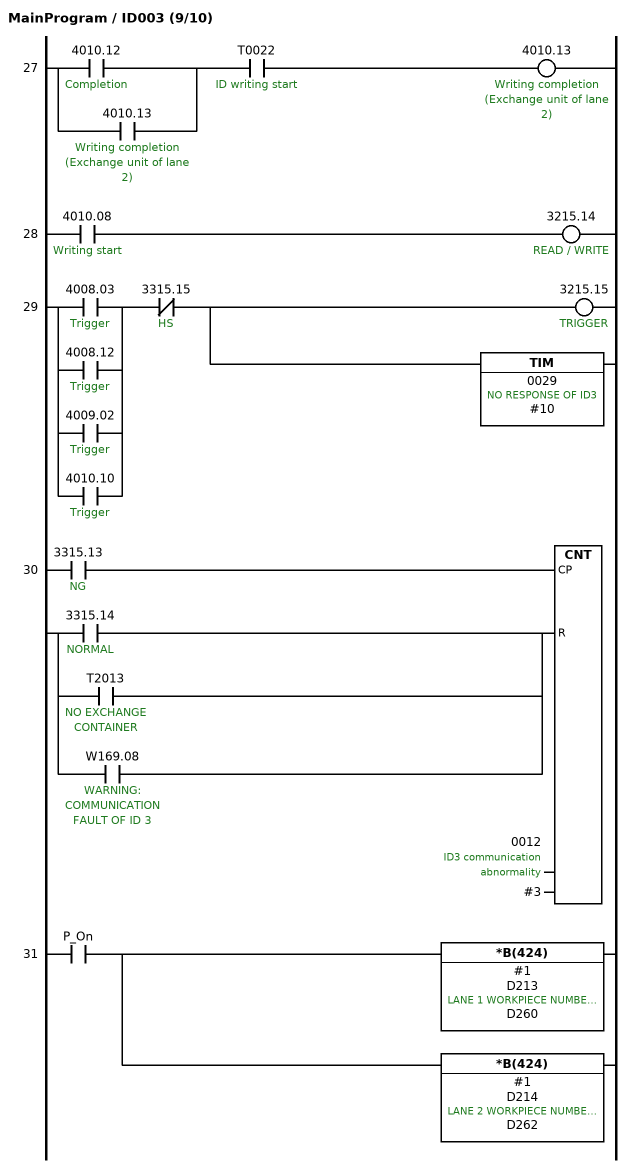
; [picture p48: MainProgram / ID003, rungs 27-31]
; rung 27
LD 4010.12  ; Completion
OR 4010.13  ; Writing completion (Exchange unit of lane 2)
AND T0022  ; ID writing start
OUT 4010.13  ; Writing completion (Exchange unit of lane 2)
; rung 28
LD 4010.08  ; Writing start
OUT 3215.14  ; READ / WRITE
; rung 29
LD 4008.03  ; Trigger
OR 4008.12  ; Trigger
OR 4009.02  ; Trigger
OR 4010.10  ; Trigger
ANDNOT 3315.15  ; HS
OUT 3215.15  ; TRIGGER
TIM 0029 #10  ; NO RESPONSE OF ID3
; rung 30
LD 3315.13  ; NG
LD 3315.14  ; NORMAL
OR T2013  ; NO EXCHANGE CONTAINER
OR W169.08  ; WARNING:COMMUNICATION FAULT OF ID 3
CNT 0012 #3  ; ID3 communication abnormality
; rung 31
LD P_On
*B(424) #1 D213 D260  ; LANE 1 WORKPIECE NUMBER DISPLAY
*B(424) #1 D214 D262  ; LANE 2 WORKPIECE NUMBER DISPLAY

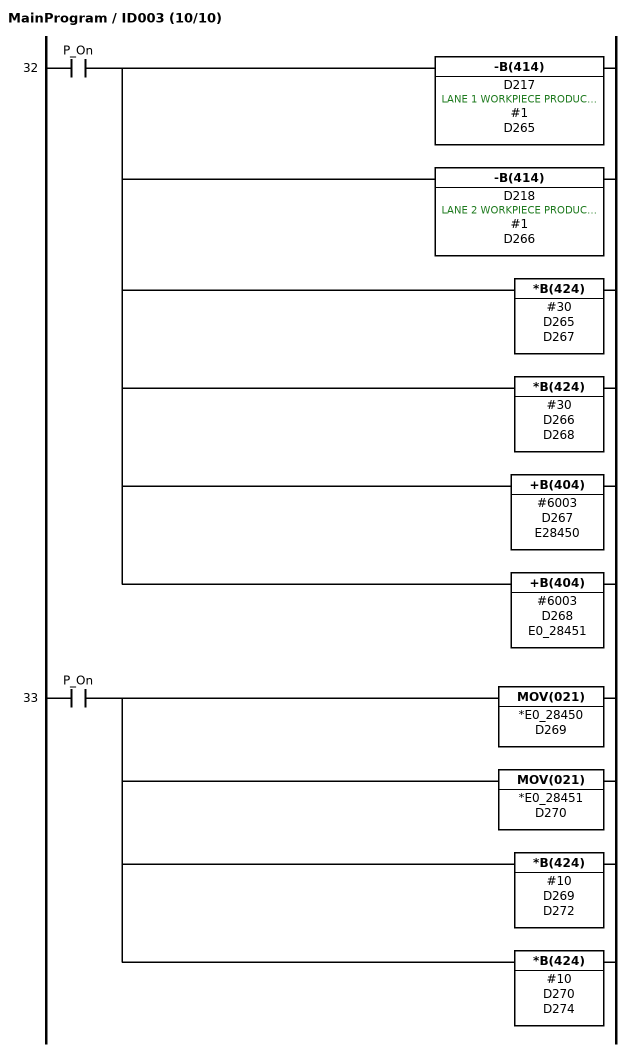
; rung 32
LD P_On
-B(414) D217 #1 D265  ; LANE 1 WORKPIECE PRODUCT NUMBER
-B(414) D218 #1 D266  ; LANE 2 WORKPIECE PRODUCT NUMBER
*B(424) #30 D265 D267
*B(424) #30 D266 D268
+B(404) #6003 D267 E28450
+B(404) #6003 D268 E0_28451
; rung 33
LD P_On
MOV(021) *E0_28450 D269
MOV(021) *E0_28451 D270
*B(424) #10 D269 D272
*B(424) #10 D270 D274

### Section ID004

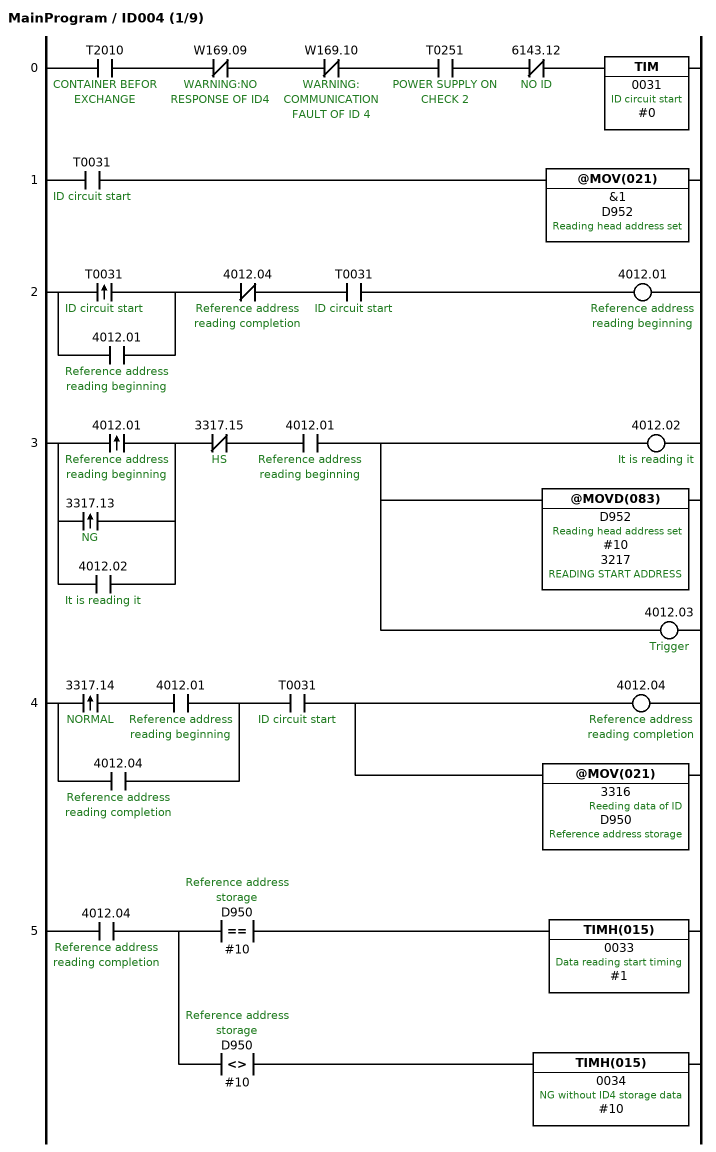
; rung 0
LD T2010  ; CONTAINER BEFOR EXCHANGE
ANDNOT W169.09  ; WARNING:NO RESPONSE OF ID4
ANDNOT W169.10  ; WARNING:COMMUNICATION FAULT OF ID 4
AND T0251  ; POWER SUPPLY ON CHECK 2
ANDNOT 6143.12  ; NO ID
TIM 0031 #0  ; ID circuit start
; rung 1
LD T0031  ; ID circuit start
@MOV(021) &1 D952  ; Reading head address set
; rung 2
@LD T0031  ; ID circuit start
OR 4012.01  ; Reference address reading beginning
ANDNOT 4012.04  ; Reference address reading completion
AND T0031  ; ID circuit start
OUT 4012.01  ; Reference address reading beginning
; rung 3
@LD 4012.01  ; Reference address reading beginning
@OR 3317.13  ; NG
OR 4012.02  ; It is reading it
ANDNOT 3317.15  ; HS
AND 4012.01  ; Reference address reading beginning
OUT 4012.02  ; It is reading it
@MOVD(083) D952 #10 3217  ; Reading head address set, READING START ADDRESS
OUT 4012.03  ; Trigger
; rung 4
@LD 3317.14  ; NORMAL
AND 4012.01  ; Reference address reading beginning
OR 4012.04  ; Reference address reading completion
AND T0031  ; ID circuit start
OUT 4012.04  ; Reference address reading completion
@MOV(021) 3316 D950  ; Reeding data of ID, Reference address storage
; rung 5
LD 4012.04  ; Reference address reading completion
OUT TR0
AND=(300) D950 #10  ; Reference address storage
TIMH(015) 0033 #1  ; Data reading start timing
LD TR0
AND<>(305) D950 #10  ; Reference address storage
TIMH(015) 0034 #10  ; NG without ID4 storage data

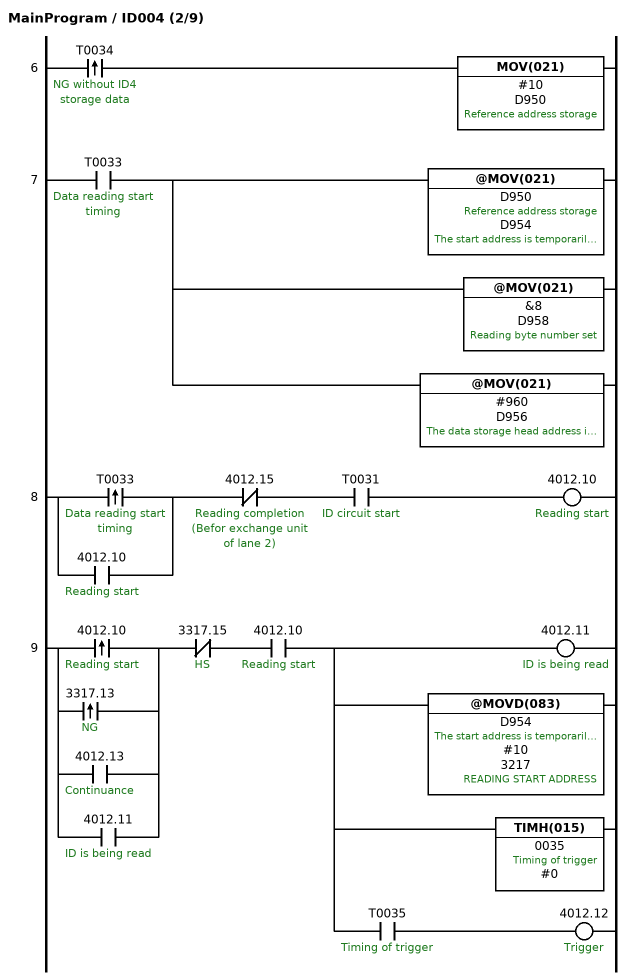
; rung 6
@LD T0034  ; NG without ID4 storage data
MOV(021) #10 D950  ; Reference address storage
; rung 7
LD T0033  ; Data reading start timing
@MOV(021) D950 D954  ; Reference address storage, The start address is temporarily memorized
@MOV(021) &8 D958  ; Reading byte number set
@MOV(021) #960 D956  ; The data storage head address is memorized
; rung 8
@LD T0033  ; Data reading start timing
OR 4012.10  ; Reading start
ANDNOT 4012.15  ; Reading completion (Befor exchange unit of lane 2)
AND T0031  ; ID circuit start
OUT 4012.10  ; Reading start
; rung 9
@LD 4012.10  ; Reading start
@OR 3317.13  ; NG
OR 4012.13  ; Continuance
OR 4012.11  ; ID is being read
ANDNOT 3317.15  ; HS
AND 4012.10  ; Reading start
OUT 4012.11  ; ID is being read
@MOVD(083) D954 #10 3217  ; The start address is temporarily memorized, READING START ADDRESS
TIMH(015) 0035 #0  ; Timing of trigger
AND T0035  ; Timing of trigger
OUT 4012.12  ; Trigger

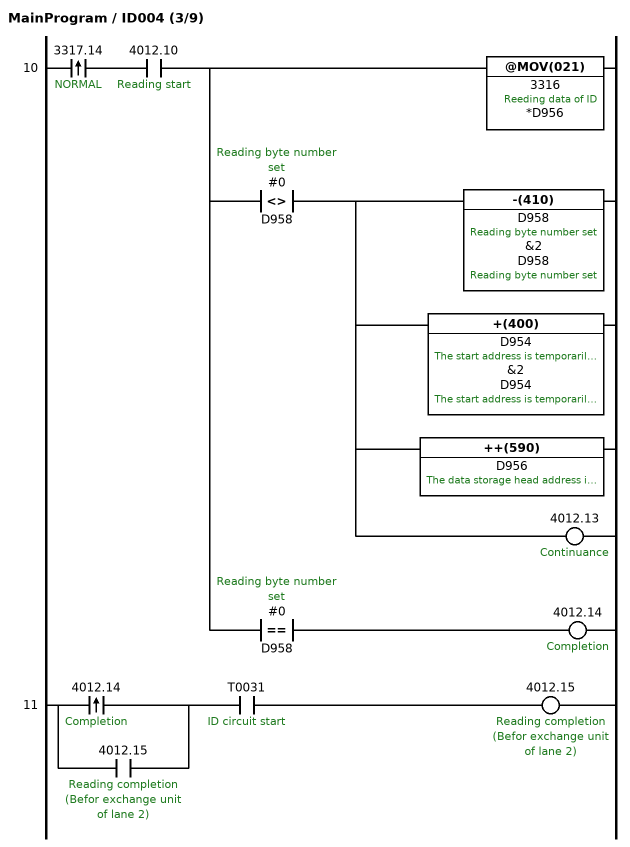
; rung 10
@LD 3317.14  ; NORMAL
AND 4012.10  ; Reading start
OUT TR0
@MOV(021) 3316 *D956  ; Reeding data of ID
AND<>(305) #0 D958  ; Reading byte number set
-(410) D958 &2 D958  ; Reading byte number set
+(400) D954 &2 D954  ; The start address is temporarily memorized
++(590) D956  ; The data storage head address is memorized
OUT 4012.13  ; Continuance
LD TR0
AND=(300) #0 D958  ; Reading byte number set
OUT 4012.14  ; Completion
; rung 11
@LD 4012.14  ; Completion
OR 4012.15  ; Reading completion (Befor exchange unit of lane 2)
AND T0031  ; ID circuit start
OUT 4012.15  ; Reading completion (Befor exchange unit of lane 2)

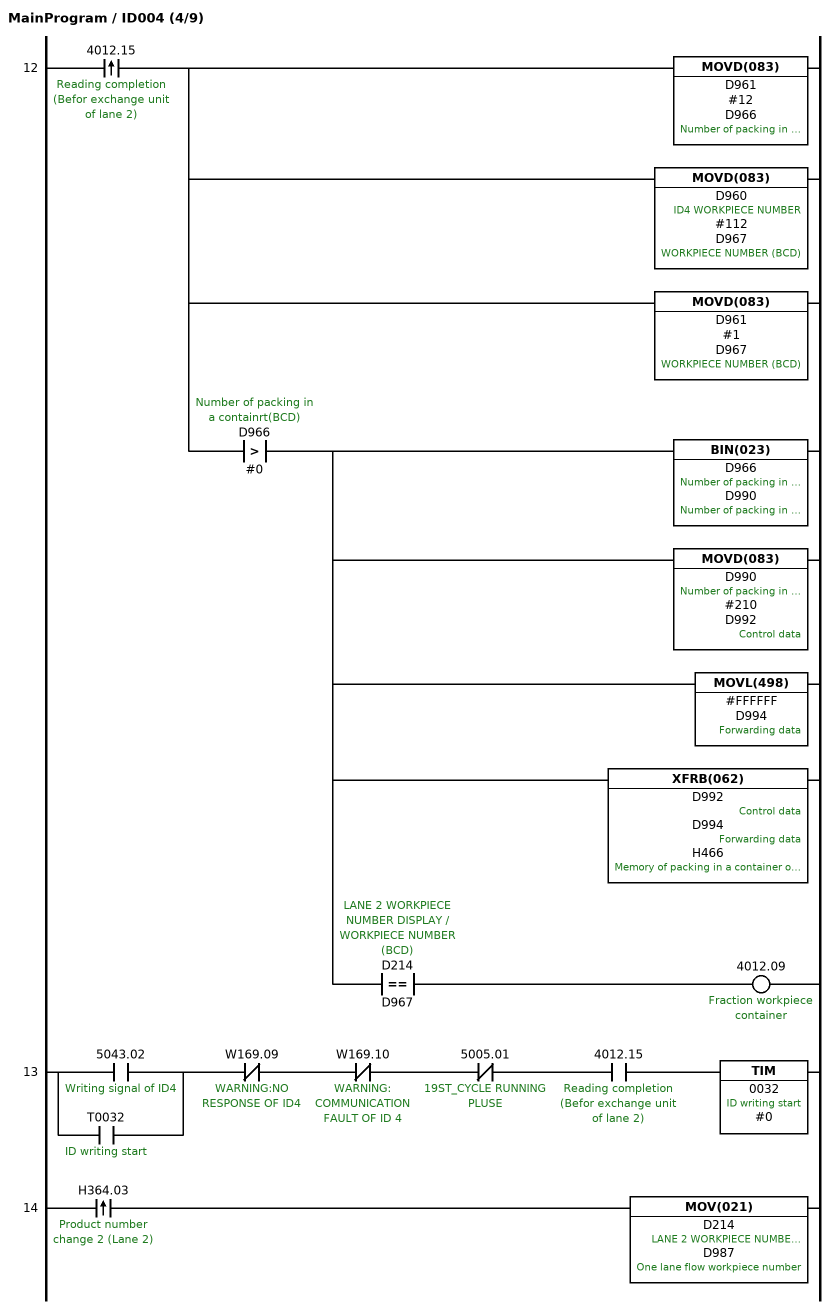
; rung 12
@LD 4012.15  ; Reading completion (Befor exchange unit of lane 2)
MOVD(083) D961 #12 D966  ; Number of packing in a containrt(BCD)
MOVD(083) D960 #112 D967  ; ID4 WORKPIECE NUMBER, WORKPIECE NUMBER (BCD)
MOVD(083) D961 #1 D967  ; WORKPIECE NUMBER (BCD)
AND>(320) D966 #0  ; Number of packing in a containrt(BCD)
BIN(023) D966 D990  ; Number of packing in a containrt(BCD), Number of packing in a containrt(BIN)
MOVD(083) D990 #210 D992  ; Number of packing in a containrt(BIN), Control data
MOVL(498) #FFFFFF D994  ; Forwarding data
XFRB(062) D992 D994 H466  ; Control data, Forwarding data, Memory of packing in a container of lane 2 (container befor exchange)
AND=(300) D214 D967  ; LANE 2 WORKPIECE NUMBER DISPLAY, WORKPIECE NUMBER (BCD)
OUT 4012.09  ; Fraction workpiece container
; rung 13
LD 5043.02  ; Writing signal of ID4
OR T0032  ; ID writing start
ANDNOT W169.09  ; WARNING:NO RESPONSE OF ID4
ANDNOT W169.10  ; WARNING:COMMUNICATION FAULT OF ID 4
ANDNOT 5005.01  ; 19ST_CYCLE RUNNING PLUSE
AND 4012.15  ; Reading completion (Befor exchange unit of lane 2)
TIM 0032 #0  ; ID writing start
; rung 14
@LD H364.03  ; Product number change 2 (Lane 2)
MOV(021) D214 D987  ; LANE 2 WORKPIECE NUMBER DISPLAY, One lane flow workpiece number

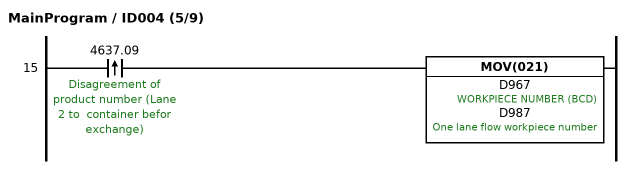
; rung 15
@LD 4637.09  ; Disagreement of product number (Lane 2 to  container befor exchange)
MOV(021) D967 D987  ; WORKPIECE NUMBER (BCD), One lane flow workpiece number

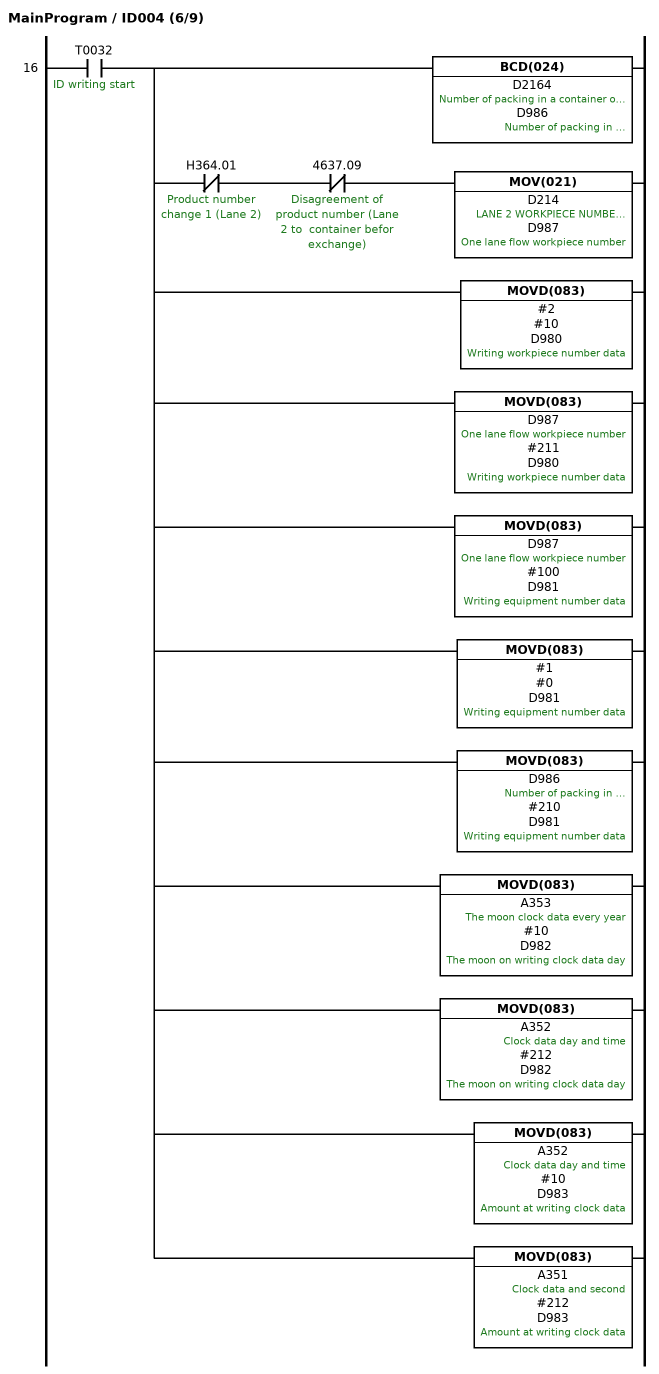
; rung 16
LD T0032  ; ID writing start
OUT TR0
BCD(024) D2164 D986  ; Number of packing in a container of lane 2 (container before exchange)(BIN), Number of packing in a containrt(BCD)
ANDNOT H364.01  ; Product number change 1 (Lane 2)
ANDNOT 4637.09  ; Disagreement of product number (Lane 2 to  container befor exchange)
MOV(021) D214 D987  ; LANE 2 WORKPIECE NUMBER DISPLAY, One lane flow workpiece number
LD TR0
MOVD(083) #2 #10 D980  ; Writing workpiece number data
MOVD(083) D987 #211 D980  ; One lane flow workpiece number, Writing workpiece number data
MOVD(083) D987 #100 D981  ; One lane flow workpiece number, Writing equipment number data
MOVD(083) #1 #0 D981  ; Writing equipment number data
MOVD(083) D986 #210 D981  ; Number of packing in a containrt(BCD), Writing equipment number data
MOVD(083) A353 #10 D982  ; The moon clock data every year, The moon on writing clock data day
MOVD(083) A352 #212 D982  ; Clock data day and time, The moon on writing clock data day
MOVD(083) A352 #10 D983  ; Clock data day and time, Amount at writing clock data
MOVD(083) A351 #212 D983  ; Clock data and second, Amount at writing clock data

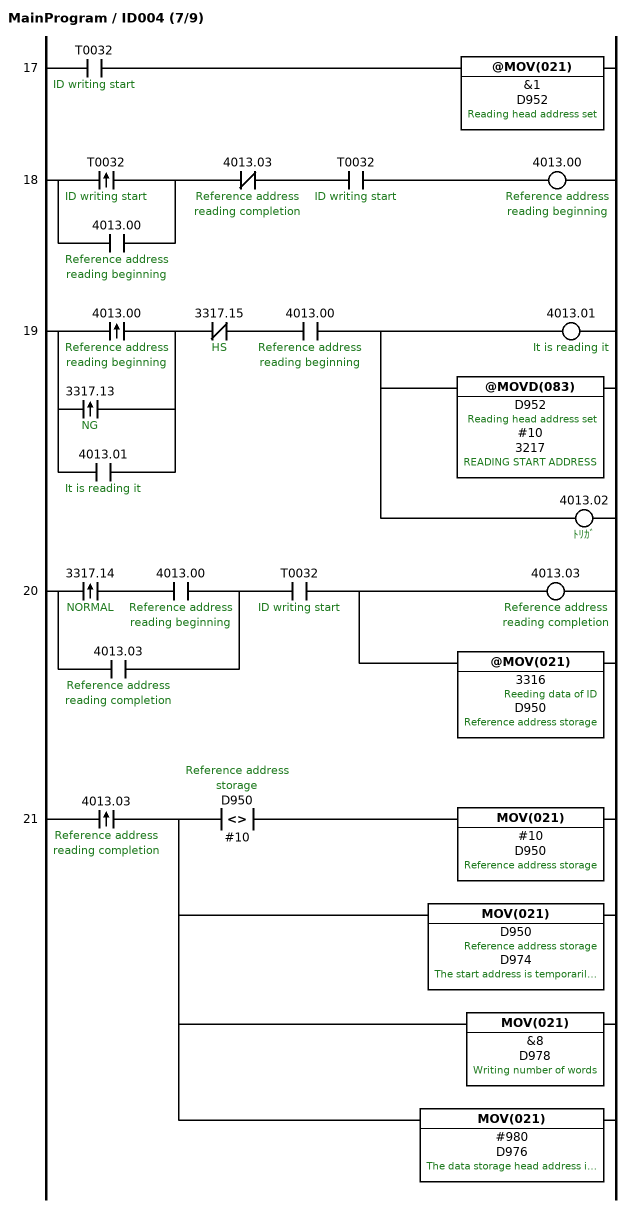
; rung 17
LD T0032  ; ID writing start
@MOV(021) &1 D952  ; Reading head address set
; rung 18
@LD T0032  ; ID writing start
OR 4013.00  ; Reference address reading beginning
ANDNOT 4013.03  ; Reference address reading completion
AND T0032  ; ID writing start
OUT 4013.00  ; Reference address reading beginning
; rung 19
@LD 4013.00  ; Reference address reading beginning
@OR 3317.13  ; NG
OR 4013.01  ; It is reading it
ANDNOT 3317.15  ; HS
AND 4013.00  ; Reference address reading beginning
OUT 4013.01  ; It is reading it
@MOVD(083) D952 #10 3217  ; Reading head address set, READING START ADDRESS
OUT 4013.02  ; ﾄﾘｶﾞ
; rung 20
@LD 3317.14  ; NORMAL
AND 4013.00  ; Reference address reading beginning
OR 4013.03  ; Reference address reading completion
AND T0032  ; ID writing start
OUT 4013.03  ; Reference address reading completion
@MOV(021) 3316 D950  ; Reeding data of ID, Reference address storage
; rung 21
@LD 4013.03  ; Reference address reading completion
OUT TR0
AND<>(305) D950 #10  ; Reference address storage
MOV(021) #10 D950  ; Reference address storage
LD TR0
MOV(021) D950 D974  ; Reference address storage, The start address is temporarily memorized
MOV(021) &8 D978  ; Writing number of words
MOV(021) #980 D976  ; The data storage head address is memorized

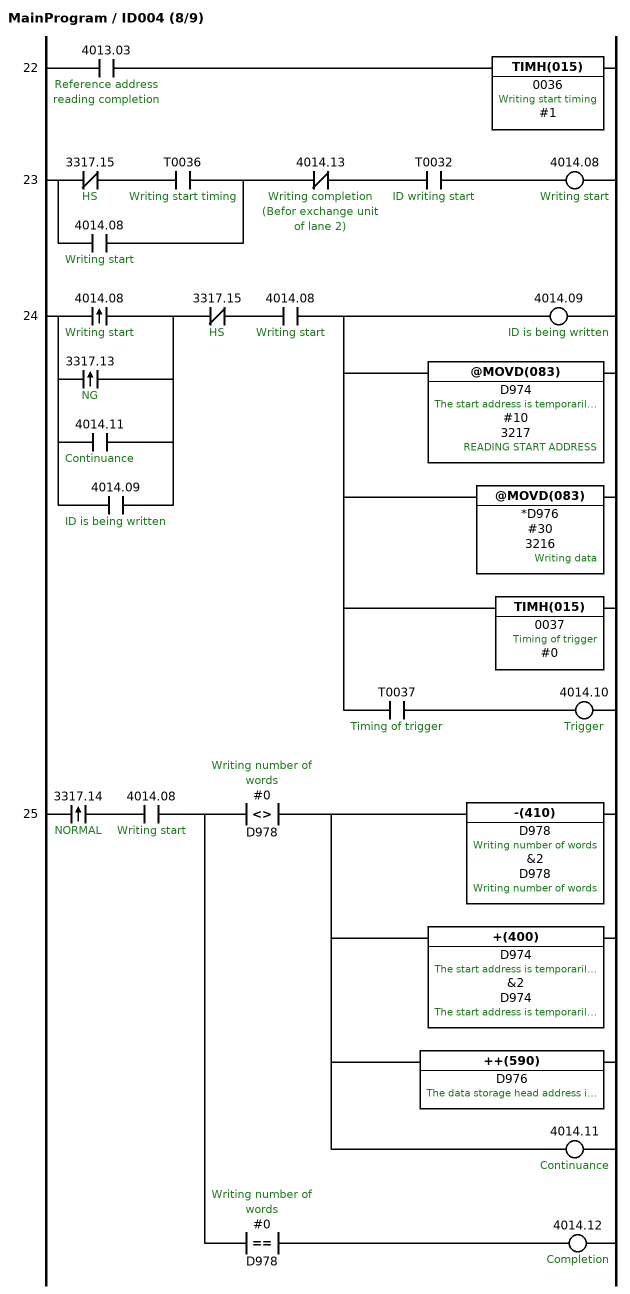
; rung 22
LD 4013.03  ; Reference address reading completion
TIMH(015) 0036 #1  ; Writing start timing
; rung 23
LDNOT 3317.15  ; HS
AND T0036  ; Writing start timing
OR 4014.08  ; Writing start
ANDNOT 4014.13  ; Writing completion (Befor exchange unit of lane 2)
AND T0032  ; ID writing start
OUT 4014.08  ; Writing start
; rung 24
@LD 4014.08  ; Writing start
@OR 3317.13  ; NG
OR 4014.11  ; Continuance
OR 4014.09  ; ID is being written
ANDNOT 3317.15  ; HS
AND 4014.08  ; Writing start
OUT 4014.09  ; ID is being written
@MOVD(083) D974 #10 3217  ; The start address is temporarily memorized, READING START ADDRESS
@MOVD(083) *D976 #30 3216  ; Writing data
TIMH(015) 0037 #0  ; Timing of trigger
AND T0037  ; Timing of trigger
OUT 4014.10  ; Trigger
; rung 25
@LD 3317.14  ; NORMAL
AND 4014.08  ; Writing start
OUT TR0
AND<>(305) #0 D978  ; Writing number of words
-(410) D978 &2 D978  ; Writing number of words
+(400) D974 &2 D974  ; The start address is temporarily memorized
++(590) D976  ; The data storage head address is memorized
OUT 4014.11  ; Continuance
LD TR0
AND=(300) #0 D978  ; Writing number of words
OUT 4014.12  ; Completion

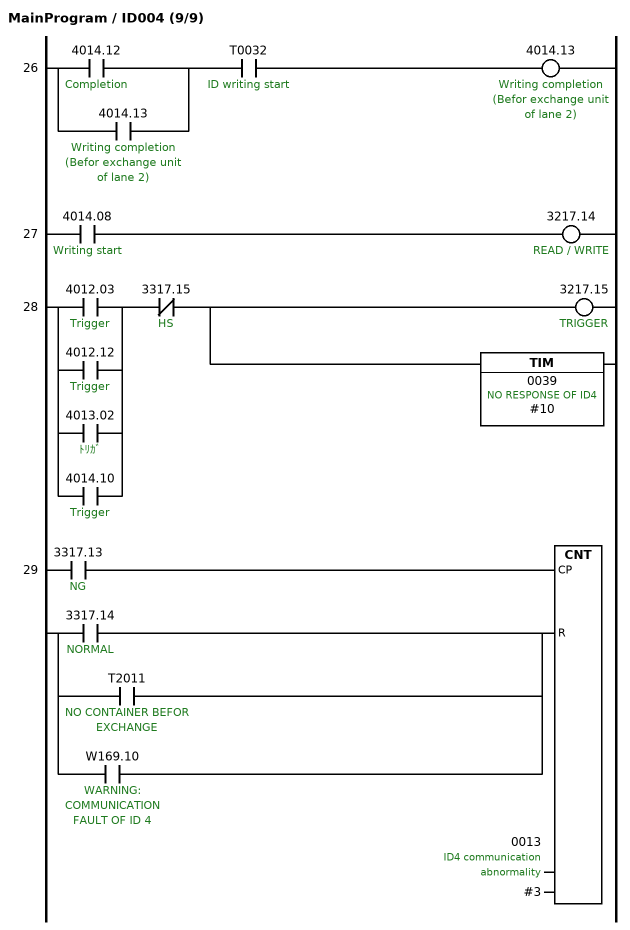
; rung 26
LD 4014.12  ; Completion
OR 4014.13  ; Writing completion (Befor exchange unit of lane 2)
AND T0032  ; ID writing start
OUT 4014.13  ; Writing completion (Befor exchange unit of lane 2)
; rung 27
LD 4014.08  ; Writing start
OUT 3217.14  ; READ / WRITE
; rung 28
LD 4012.03  ; Trigger
OR 4012.12  ; Trigger
OR 4013.02  ; ﾄﾘｶﾞ
OR 4014.10  ; Trigger
ANDNOT 3317.15  ; HS
OUT 3217.15  ; TRIGGER
TIM 0039 #10  ; NO RESPONSE OF ID4
; rung 29
LD 3317.13  ; NG
LD 3317.14  ; NORMAL
OR T2011  ; NO CONTAINER BEFOR EXCHANGE
OR W169.10  ; WARNING:COMMUNICATION FAULT OF ID 4
CNT 0013 #3  ; ID4 communication abnormality

### Section DISPLAY_CONTROL

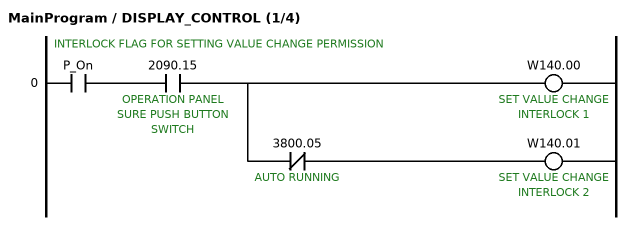
; rung 0: INTERLOCK FLAG FOR SETTING VALUE CHANGE PERMISSION
LD P_On
AND 2090.15  ; OPERATION PANEL SURE PUSH BUTTON SWITCH
OUT W140.00  ; SET VALUE CHANGE INTERLOCK 1
ANDNOT 3800.05  ; AUTO RUNNING
OUT W140.01  ; SET VALUE CHANGE INTERLOCK 2

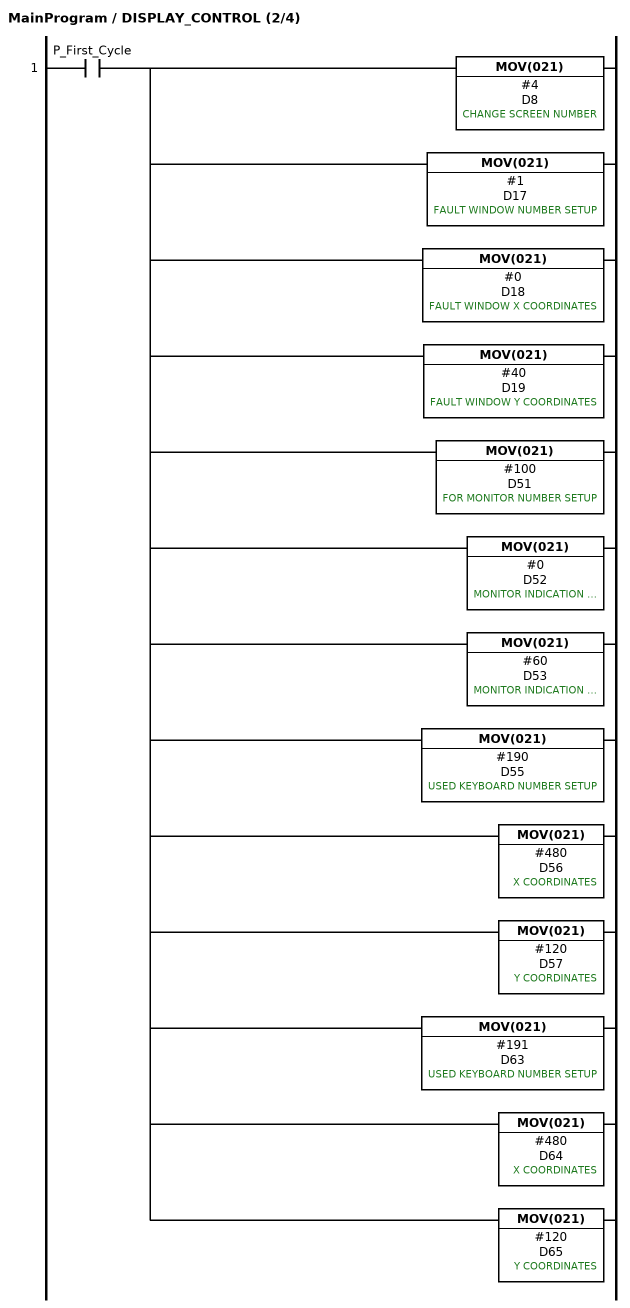
; rung 1
LD P_First_Cycle
MOV(021) #4 D8  ; CHANGE SCREEN NUMBER  // Screen number
MOV(021) #1 D17  ; FAULT WINDOW NUMBER SETUP  // Fault page screen number
MOV(021) #0 D18  ; FAULT WINDOW X COORDINATES  // Fault display position X-coordinates transmission
MOV(021) #40 D19  ; FAULT WINDOW Y COORDINATES  // Fault display position Y-coordinates transmission
MOV(021) #100 D51  ; FOR MONITOR NUMBER SETUP  // Monitor screen number
MOV(021) #0 D52  ; MONITOR INDICATION X COORDINATES  // Monitor display position X-coordinates transmission
MOV(021) #60 D53  ; MONITOR INDICATION Y COORDINATES  // Monitor display position Y-coordinates transmission
MOV(021) #190 D55  ; USED KEYBOARD NUMBER SETUP  // BCD keyboard number
MOV(021) #480 D56  ; X COORDINATES
MOV(021) #120 D57  ; Y COORDINATES
MOV(021) #191 D63  ; USED KEYBOARD NUMBER SETUP  // BIN keyboard number
MOV(021) #480 D64  ; X COORDINATES
MOV(021) #120 D65  ; Y COORDINATES

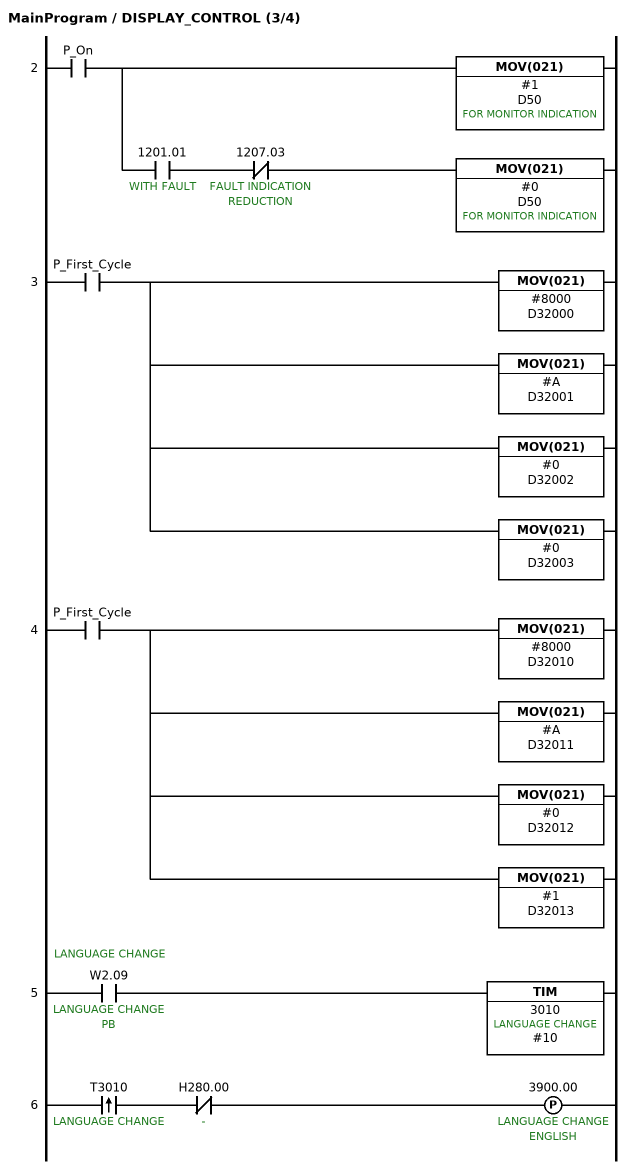
; rung 2
LD P_On
MOV(021) #1 D50  ; FOR MONITOR INDICATION  // Constant transmission with monitor display
AND 1201.01  ; WITH FAULT
ANDNOT 1207.03  ; FAULT INDICATION REDUCTION
MOV(021) #0 D50  ; FOR MONITOR INDICATION  // Monitor display overlap prevents to fault display
; rung 3
LD P_First_Cycle
MOV(021) #8000 D32000  // Arbitrary setting, start 1bit, data 7bit, stop 2bit, and even number of parity
MOV(021) #A D32001  // Transmission speed: 115200bps
MOV(021) #0 D32002
MOV(021) #0 D32003  // The 0th high-ranking link machine
; rung 4
LD P_First_Cycle
MOV(021) #8000 D32010  // Arbitrary setting, start 1bit, data 7bit, stop 2bit, and even number of parity
MOV(021) #A D32011  // Transmission speed: 115200bps
MOV(021) #0 D32012
MOV(021) #1 D32013  // The 1th high-ranking link machine
; rung 5: LANGUAGE CHANGE
LD W2.09  ; LANGUAGE CHANGE PB
TIM 3010 #10  ; LANGUAGE CHANGE
; rung 6
@LD T3010  ; LANGUAGE CHANGE
ANDNOT H280.00  ; -
DIFU(013) 3900.00  ; LANGUAGE CHANGE ENGLISH

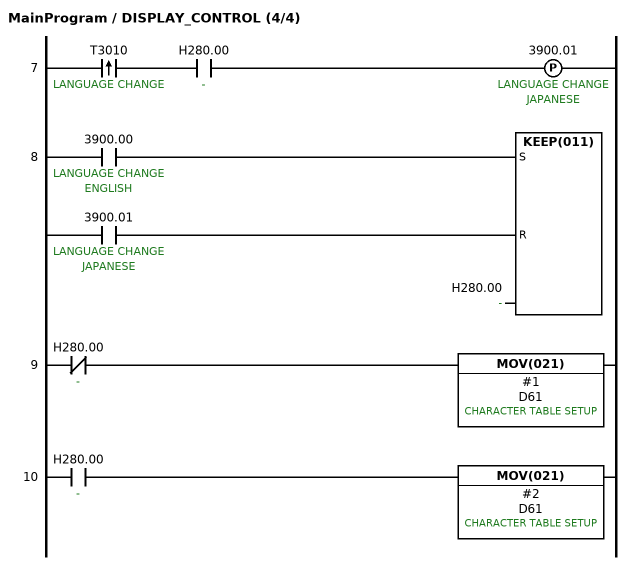
; rung 7
@LD T3010  ; LANGUAGE CHANGE
AND H280.00  ; -
DIFU(013) 3900.01  ; LANGUAGE CHANGE JAPANESE
; rung 8
LD 3900.00  ; LANGUAGE CHANGE ENGLISH
LD 3900.01  ; LANGUAGE CHANGE JAPANESE
KEEP(011) H280.00  ; -
; rung 9
LDNOT H280.00  ; -
MOV(021) #1 D61  ; CHARACTER TABLE SETUP
; rung 10
LD H280.00  ; -
MOV(021) #2 D61  ; CHARACTER TABLE SETUP

### Section FAULT

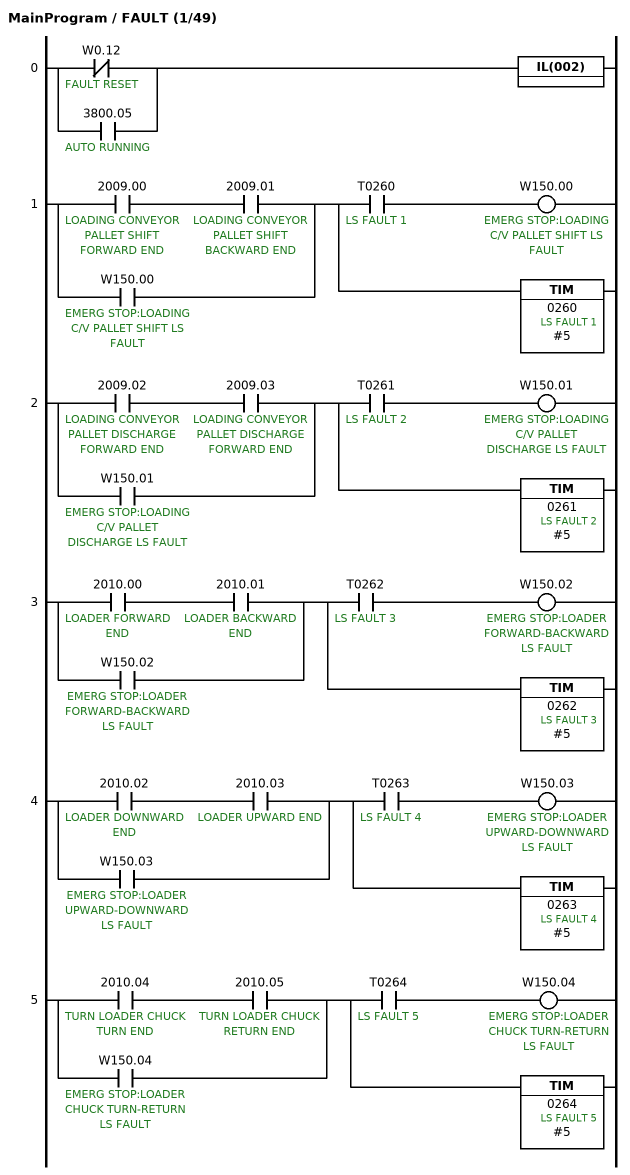
; rung 0
LDNOT W0.12  ; FAULT RESET
OR 3800.05  ; AUTO RUNNING
IL(002)
; rung 1
LD 2009.00  ; LOADING CONVEYOR PALLET SHIFT FORWARD END
AND 2009.01  ; LOADING CONVEYOR PALLET SHIFT BACKWARD END
OR W150.00  ; EMERG STOP:LOADING C/V PALLET SHIFT LS FAULT
OUT TR0
AND T0260  ; LS FAULT 1
OUT W150.00  ; EMERG STOP:LOADING C/V PALLET SHIFT LS FAULT
LD TR0
TIM 0260 #5  ; LS FAULT 1
; rung 2
LD 2009.02  ; LOADING CONVEYOR PALLET DISCHARGE FORWARD END
AND 2009.03  ; LOADING CONVEYOR PALLET DISCHARGE FORWARD END
OR W150.01  ; EMERG STOP:LOADING C/V PALLET DISCHARGE LS FAULT
OUT TR0
AND T0261  ; LS FAULT 2
OUT W150.01  ; EMERG STOP:LOADING C/V PALLET DISCHARGE LS FAULT
LD TR0
TIM 0261 #5  ; LS FAULT 2
; rung 3
LD 2010.00  ; LOADER FORWARD END
AND 2010.01  ; LOADER BACKWARD END
OR W150.02  ; EMERG STOP:LOADER FORWARD-BACKWARD LS FAULT
OUT TR0
AND T0262  ; LS FAULT 3
OUT W150.02  ; EMERG STOP:LOADER FORWARD-BACKWARD LS FAULT
LD TR0
TIM 0262 #5  ; LS FAULT 3
; rung 4
LD 2010.02  ; LOADER DOWNWARD END
AND 2010.03  ; LOADER UPWARD END
OR W150.03  ; EMERG STOP:LOADER UPWARD-DOWNWARD LS FAULT
OUT TR0
AND T0263  ; LS FAULT 4
OUT W150.03  ; EMERG STOP:LOADER UPWARD-DOWNWARD LS FAULT
LD TR0
TIM 0263 #5  ; LS FAULT 4
; rung 5
LD 2010.04  ; TURN LOADER CHUCK TURN END
AND 2010.05  ; TURN LOADER CHUCK RETURN END
OR W150.04  ; EMERG STOP:LOADER CHUCK TURN-RETURN LS FAULT
OUT TR0
AND T0264  ; LS FAULT 5
OUT W150.04  ; EMERG STOP:LOADER CHUCK TURN-RETURN LS FAULT
LD TR0
TIM 0264 #5  ; LS FAULT 5

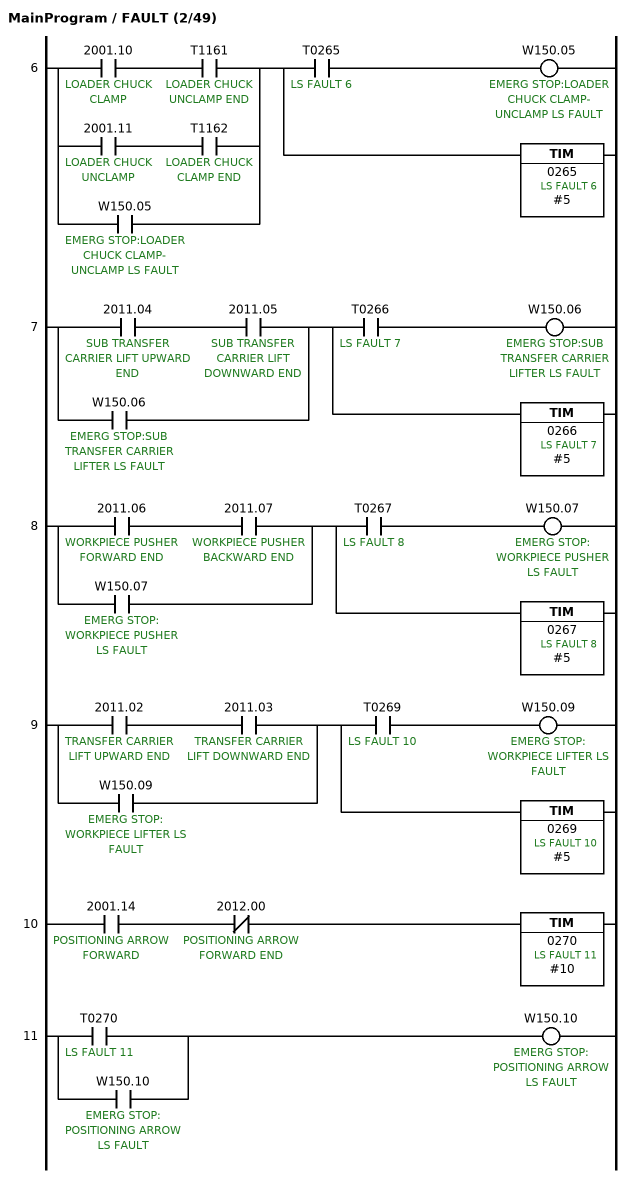
; rung 6
LD 2001.10  ; LOADER CHUCK CLAMP
AND T1161  ; LOADER CHUCK UNCLAMP END
LD 2001.11  ; LOADER CHUCK UNCLAMP
AND T1162  ; LOADER CHUCK CLAMP END
ORLD
OR W150.05  ; EMERG STOP:LOADER CHUCK CLAMP-UNCLAMP LS FAULT
OUT TR0
AND T0265  ; LS FAULT 6
OUT W150.05  ; EMERG STOP:LOADER CHUCK CLAMP-UNCLAMP LS FAULT
LD TR0
TIM 0265 #5  ; LS FAULT 6
; rung 7
LD 2011.04  ; SUB TRANSFER CARRIER LIFT UPWARD END
AND 2011.05  ; SUB TRANSFER CARRIER LIFT DOWNWARD END
OR W150.06  ; EMERG STOP:SUB TRANSFER CARRIER LIFTER LS FAULT
OUT TR0
AND T0266  ; LS FAULT 7
OUT W150.06  ; EMERG STOP:SUB TRANSFER CARRIER LIFTER LS FAULT
LD TR0
TIM 0266 #5  ; LS FAULT 7
; rung 8
LD 2011.06  ; WORKPIECE PUSHER FORWARD END
AND 2011.07  ; WORKPIECE PUSHER BACKWARD END
OR W150.07  ; EMERG STOP:WORKPIECE PUSHER LS FAULT
OUT TR0
AND T0267  ; LS FAULT 8
OUT W150.07  ; EMERG STOP:WORKPIECE PUSHER LS FAULT
LD TR0
TIM 0267 #5  ; LS FAULT 8
; rung 9
LD 2011.02  ; TRANSFER CARRIER LIFT UPWARD END
AND 2011.03  ; TRANSFER CARRIER LIFT DOWNWARD END
OR W150.09  ; EMERG STOP:WORKPIECE LIFTER LS FAULT
OUT TR0
AND T0269  ; LS FAULT 10
OUT W150.09  ; EMERG STOP:WORKPIECE LIFTER LS FAULT
LD TR0
TIM 0269 #5  ; LS FAULT 10
; rung 10
LD 2001.14  ; POSITIONING ARROW FORWARD
ANDNOT 2012.00  ; POSITIONING ARROW FORWARD END
TIM 0270 #10  ; LS FAULT 11
; rung 11
LD T0270  ; LS FAULT 11
OR W150.10  ; EMERG STOP:POSITIONING ARROW LS FAULT
OUT W150.10  ; EMERG STOP:POSITIONING ARROW LS FAULT

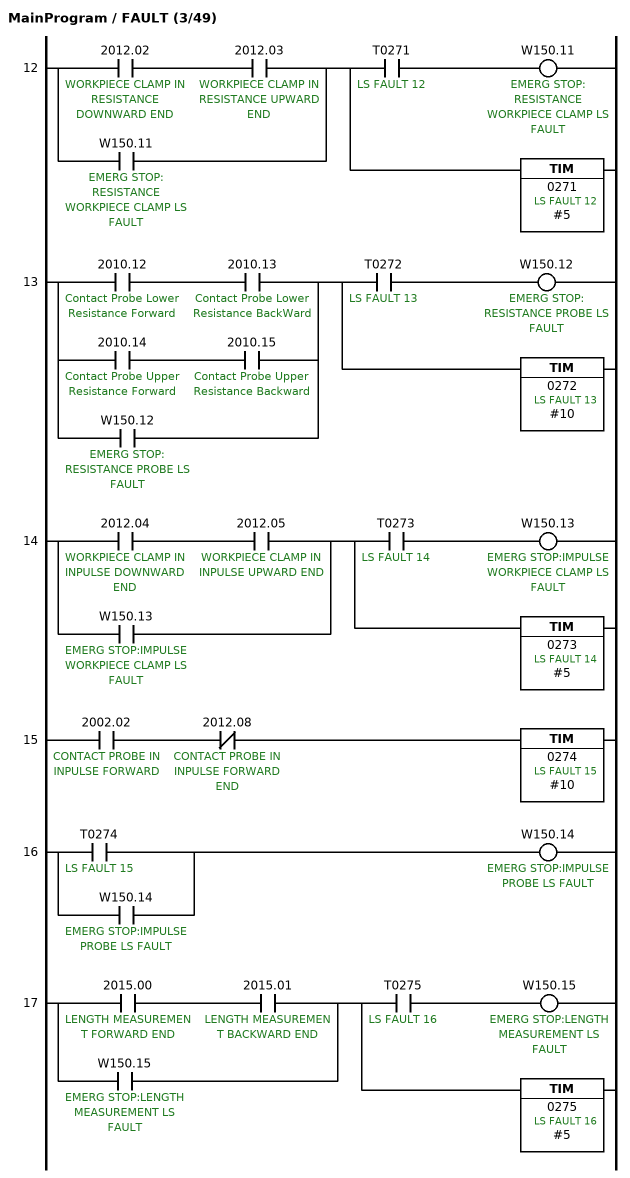
; rung 12
LD 2012.02  ; WORKPIECE CLAMP IN RESISTANCE DOWNWARD END
AND 2012.03  ; WORKPIECE CLAMP IN RESISTANCE UPWARD END
OR W150.11  ; EMERG STOP:RESISTANCE WORKPIECE CLAMP LS FAULT
OUT TR0
AND T0271  ; LS FAULT 12
OUT W150.11  ; EMERG STOP:RESISTANCE WORKPIECE CLAMP LS FAULT
LD TR0
TIM 0271 #5  ; LS FAULT 12
; rung 13
LD 2010.12  ; Contact Probe Lower Resistance Forward
AND 2010.13  ; Contact Probe Lower Resistance BackWard
LD 2010.14  ; Contact Probe Upper Resistance Forward
AND 2010.15  ; Contact Probe Upper Resistance Backward
ORLD
OR W150.12  ; EMERG STOP:RESISTANCE PROBE LS FAULT
OUT TR0
AND T0272  ; LS FAULT 13
OUT W150.12  ; EMERG STOP:RESISTANCE PROBE LS FAULT
LD TR0
TIM 0272 #10  ; LS FAULT 13
; rung 14
LD 2012.04  ; WORKPIECE CLAMP IN INPULSE DOWNWARD END
AND 2012.05  ; WORKPIECE CLAMP IN INPULSE UPWARD END
OR W150.13  ; EMERG STOP:IMPULSE WORKPIECE CLAMP LS FAULT
OUT TR0
AND T0273  ; LS FAULT 14
OUT W150.13  ; EMERG STOP:IMPULSE WORKPIECE CLAMP LS FAULT
LD TR0
TIM 0273 #5  ; LS FAULT 14
; rung 15
LD 2002.02  ; CONTACT PROBE IN INPULSE FORWARD
ANDNOT 2012.08  ; CONTACT PROBE IN INPULSE FORWARD END
TIM 0274 #10  ; LS FAULT 15
; rung 16
LD T0274  ; LS FAULT 15
OR W150.14  ; EMERG STOP:IMPULSE PROBE LS FAULT
OUT W150.14  ; EMERG STOP:IMPULSE PROBE LS FAULT
; rung 17
LD 2015.00  ; LENGTH MEASUREMENT FORWARD END
AND 2015.01  ; LENGTH MEASUREMENT BACKWARD END
OR W150.15  ; EMERG STOP:LENGTH MEASUREMENT LS FAULT
OUT TR0
AND T0275  ; LS FAULT 16
OUT W150.15  ; EMERG STOP:LENGTH MEASUREMENT LS FAULT
LD TR0
TIM 0275 #5  ; LS FAULT 16

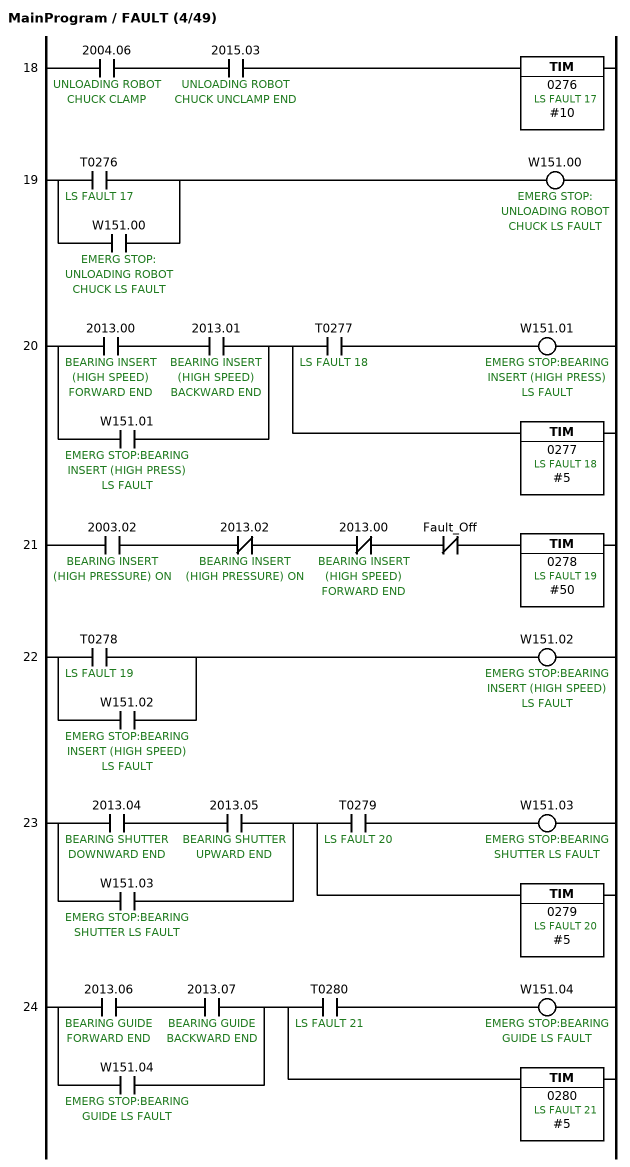
; rung 18
LD 2004.06  ; UNLOADING ROBOT CHUCK CLAMP
AND 2015.03  ; UNLOADING ROBOT CHUCK UNCLAMP END
TIM 0276 #10  ; LS FAULT 17
; rung 19
LD T0276  ; LS FAULT 17
OR W151.00  ; EMERG STOP:UNLOADING ROBOT CHUCK LS FAULT
OUT W151.00  ; EMERG STOP:UNLOADING ROBOT CHUCK LS FAULT
; rung 20
LD 2013.00  ; BEARING INSERT (HIGH SPEED) FORWARD END
AND 2013.01  ; BEARING INSERT (HIGH SPEED) BACKWARD END
OR W151.01  ; EMERG STOP:BEARING INSERT (HIGH PRESS) LS FAULT
OUT TR0
AND T0277  ; LS FAULT 18
OUT W151.01  ; EMERG STOP:BEARING INSERT (HIGH PRESS) LS FAULT
LD TR0
TIM 0277 #5  ; LS FAULT 18
; rung 21
LD 2003.02  ; BEARING INSERT (HIGH PRESSURE) ON
ANDNOT 2013.02  ; BEARING INSERT (HIGH PRESSURE) ON
ANDNOT 2013.00  ; BEARING INSERT (HIGH SPEED) FORWARD END
ANDNOT Fault_Off
TIM 0278 #50  ; LS FAULT 19
; rung 22
LD T0278  ; LS FAULT 19
OR W151.02  ; EMERG STOP:BEARING INSERT (HIGH SPEED) LS FAULT
OUT W151.02  ; EMERG STOP:BEARING INSERT (HIGH SPEED) LS FAULT
; rung 23
LD 2013.04  ; BEARING SHUTTER DOWNWARD END
AND 2013.05  ; BEARING SHUTTER UPWARD END
OR W151.03  ; EMERG STOP:BEARING SHUTTER LS FAULT
OUT TR0
AND T0279  ; LS FAULT 20
OUT W151.03  ; EMERG STOP:BEARING SHUTTER LS FAULT
LD TR0
TIM 0279 #5  ; LS FAULT 20
; rung 24
LD 2013.06  ; BEARING GUIDE FORWARD END
AND 2013.07  ; BEARING GUIDE BACKWARD END
OR W151.04  ; EMERG STOP:BEARING GUIDE LS FAULT
OUT TR0
AND T0280  ; LS FAULT 21
OUT W151.04  ; EMERG STOP:BEARING GUIDE LS FAULT
LD TR0
TIM 0280 #5  ; LS FAULT 21

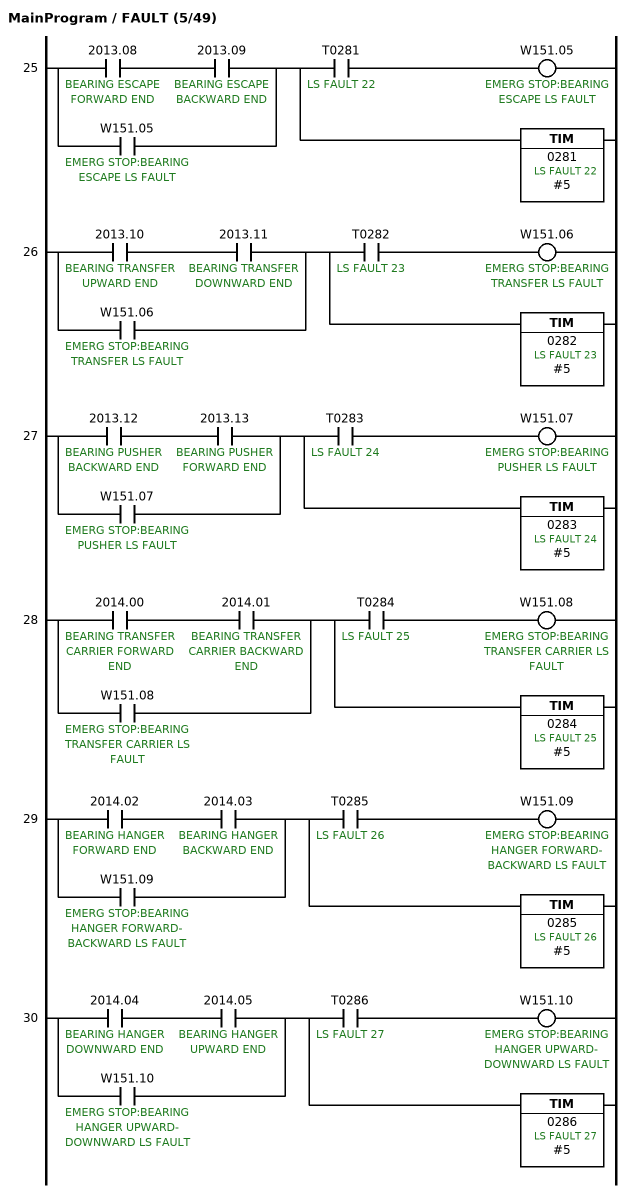
; rung 25
LD 2013.08  ; BEARING ESCAPE FORWARD END
AND 2013.09  ; BEARING ESCAPE BACKWARD END
OR W151.05  ; EMERG STOP:BEARING ESCAPE LS FAULT
OUT TR0
AND T0281  ; LS FAULT 22
OUT W151.05  ; EMERG STOP:BEARING ESCAPE LS FAULT
LD TR0
TIM 0281 #5  ; LS FAULT 22
; rung 26
LD 2013.10  ; BEARING TRANSFER UPWARD END
AND 2013.11  ; BEARING TRANSFER DOWNWARD END
OR W151.06  ; EMERG STOP:BEARING TRANSFER LS FAULT
OUT TR0
AND T0282  ; LS FAULT 23
OUT W151.06  ; EMERG STOP:BEARING TRANSFER LS FAULT
LD TR0
TIM 0282 #5  ; LS FAULT 23
; rung 27
LD 2013.12  ; BEARING PUSHER BACKWARD END
AND 2013.13  ; BEARING PUSHER FORWARD END
OR W151.07  ; EMERG STOP:BEARING PUSHER LS FAULT
OUT TR0
AND T0283  ; LS FAULT 24
OUT W151.07  ; EMERG STOP:BEARING PUSHER LS FAULT
LD TR0
TIM 0283 #5  ; LS FAULT 24
; rung 28
LD 2014.00  ; BEARING TRANSFER CARRIER FORWARD END
AND 2014.01  ; BEARING TRANSFER CARRIER BACKWARD END
OR W151.08  ; EMERG STOP:BEARING TRANSFER CARRIER LS FAULT
OUT TR0
AND T0284  ; LS FAULT 25
OUT W151.08  ; EMERG STOP:BEARING TRANSFER CARRIER LS FAULT
LD TR0
TIM 0284 #5  ; LS FAULT 25
; rung 29
LD 2014.02  ; BEARING HANGER FORWARD END
AND 2014.03  ; BEARING HANGER BACKWARD END
OR W151.09  ; EMERG STOP:BEARING HANGER FORWARD-BACKWARD LS FAULT
OUT TR0
AND T0285  ; LS FAULT 26
OUT W151.09  ; EMERG STOP:BEARING HANGER FORWARD-BACKWARD LS FAULT
LD TR0
TIM 0285 #5  ; LS FAULT 26
; rung 30
LD 2014.04  ; BEARING HANGER DOWNWARD END
AND 2014.05  ; BEARING HANGER UPWARD END
OR W151.10  ; EMERG STOP:BEARING HANGER UPWARD-DOWNWARD LS FAULT
OUT TR0
AND T0286  ; LS FAULT 27
OUT W151.10  ; EMERG STOP:BEARING HANGER UPWARD-DOWNWARD LS FAULT
LD TR0
TIM 0286 #5  ; LS FAULT 27

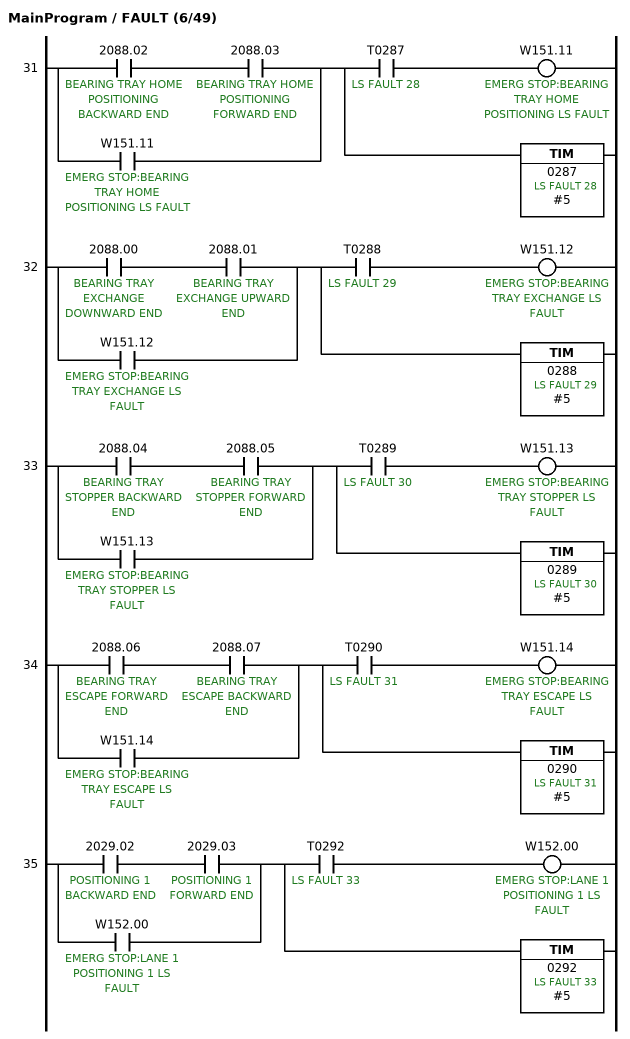
; rung 31
LD 2088.02  ; BEARING TRAY HOME POSITIONING BACKWARD END
AND 2088.03  ; BEARING TRAY HOME POSITIONING FORWARD END
OR W151.11  ; EMERG STOP:BEARING TRAY HOME POSITIONING LS FAULT
OUT TR0
AND T0287  ; LS FAULT 28
OUT W151.11  ; EMERG STOP:BEARING TRAY HOME POSITIONING LS FAULT
LD TR0
TIM 0287 #5  ; LS FAULT 28
; rung 32
LD 2088.00  ; BEARING TRAY EXCHANGE DOWNWARD END
AND 2088.01  ; BEARING TRAY EXCHANGE UPWARD END
OR W151.12  ; EMERG STOP:BEARING TRAY EXCHANGE LS FAULT
OUT TR0
AND T0288  ; LS FAULT 29
OUT W151.12  ; EMERG STOP:BEARING TRAY EXCHANGE LS FAULT
LD TR0
TIM 0288 #5  ; LS FAULT 29
; rung 33
LD 2088.04  ; BEARING TRAY STOPPER BACKWARD END
AND 2088.05  ; BEARING TRAY STOPPER FORWARD END
OR W151.13  ; EMERG STOP:BEARING TRAY STOPPER LS FAULT
OUT TR0
AND T0289  ; LS FAULT 30
OUT W151.13  ; EMERG STOP:BEARING TRAY STOPPER LS FAULT
LD TR0
TIM 0289 #5  ; LS FAULT 30
; rung 34
LD 2088.06  ; BEARING TRAY ESCAPE FORWARD END
AND 2088.07  ; BEARING TRAY ESCAPE BACKWARD END
OR W151.14  ; EMERG STOP:BEARING TRAY ESCAPE LS FAULT
OUT TR0
AND T0290  ; LS FAULT 31
OUT W151.14  ; EMERG STOP:BEARING TRAY ESCAPE LS FAULT
LD TR0
TIM 0290 #5  ; LS FAULT 31
; rung 35
LD 2029.02  ; POSITIONING 1 BACKWARD END
AND 2029.03  ; POSITIONING 1 FORWARD END
OR W152.00  ; EMERG STOP:LANE 1 POSITIONING 1 LS FAULT
OUT TR0
AND T0292  ; LS FAULT 33
OUT W152.00  ; EMERG STOP:LANE 1 POSITIONING 1 LS FAULT
LD TR0
TIM 0292 #5  ; LS FAULT 33

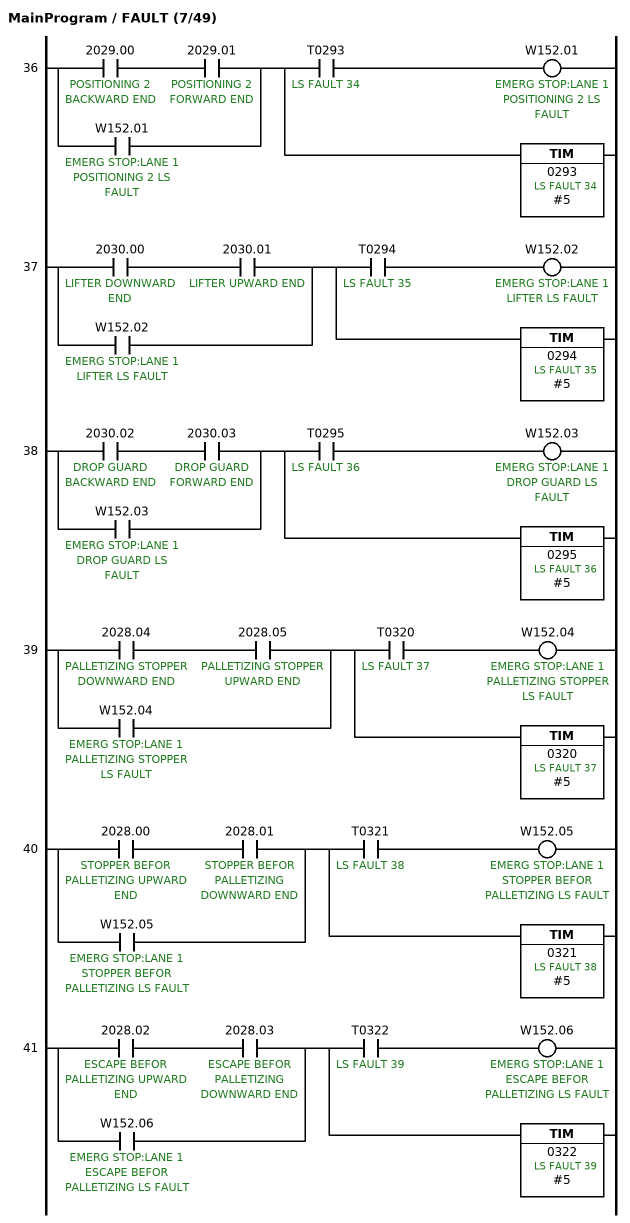
; rung 36
LD 2029.00  ; POSITIONING 2 BACKWARD END
AND 2029.01  ; POSITIONING 2 FORWARD END
OR W152.01  ; EMERG STOP:LANE 1 POSITIONING 2 LS FAULT
OUT TR0
AND T0293  ; LS FAULT 34
OUT W152.01  ; EMERG STOP:LANE 1 POSITIONING 2 LS FAULT
LD TR0
TIM 0293 #5  ; LS FAULT 34
; rung 37
LD 2030.00  ; LIFTER DOWNWARD END
AND 2030.01  ; LIFTER UPWARD END
OR W152.02  ; EMERG STOP:LANE 1 LIFTER LS FAULT
OUT TR0
AND T0294  ; LS FAULT 35
OUT W152.02  ; EMERG STOP:LANE 1 LIFTER LS FAULT
LD TR0
TIM 0294 #5  ; LS FAULT 35
; rung 38
LD 2030.02  ; DROP GUARD BACKWARD END
AND 2030.03  ; DROP GUARD FORWARD END
OR W152.03  ; EMERG STOP:LANE 1 DROP GUARD LS FAULT
OUT TR0
AND T0295  ; LS FAULT 36
OUT W152.03  ; EMERG STOP:LANE 1 DROP GUARD LS FAULT
LD TR0
TIM 0295 #5  ; LS FAULT 36
; rung 39
LD 2028.04  ; PALLETIZING STOPPER DOWNWARD END
AND 2028.05  ; PALLETIZING STOPPER UPWARD END
OR W152.04  ; EMERG STOP:LANE 1 PALLETIZING STOPPER LS FAULT
OUT TR0
AND T0320  ; LS FAULT 37
OUT W152.04  ; EMERG STOP:LANE 1 PALLETIZING STOPPER LS FAULT
LD TR0
TIM 0320 #5  ; LS FAULT 37
; rung 40
LD 2028.00  ; STOPPER BEFOR PALLETIZING UPWARD END
AND 2028.01  ; STOPPER BEFOR PALLETIZING DOWNWARD END
OR W152.05  ; EMERG STOP:LANE 1 STOPPER BEFOR PALLETIZING LS FAULT
OUT TR0
AND T0321  ; LS FAULT 38
OUT W152.05  ; EMERG STOP:LANE 1 STOPPER BEFOR PALLETIZING LS FAULT
LD TR0
TIM 0321 #5  ; LS FAULT 38
; rung 41
LD 2028.02  ; ESCAPE BEFOR PALLETIZING UPWARD END
AND 2028.03  ; ESCAPE BEFOR PALLETIZING DOWNWARD END
OR W152.06  ; EMERG STOP:LANE 1 ESCAPE BEFOR PALLETIZING LS FAULT
OUT TR0
AND T0322  ; LS FAULT 39
OUT W152.06  ; EMERG STOP:LANE 1 ESCAPE BEFOR PALLETIZING LS FAULT
LD TR0
TIM 0322 #5  ; LS FAULT 39

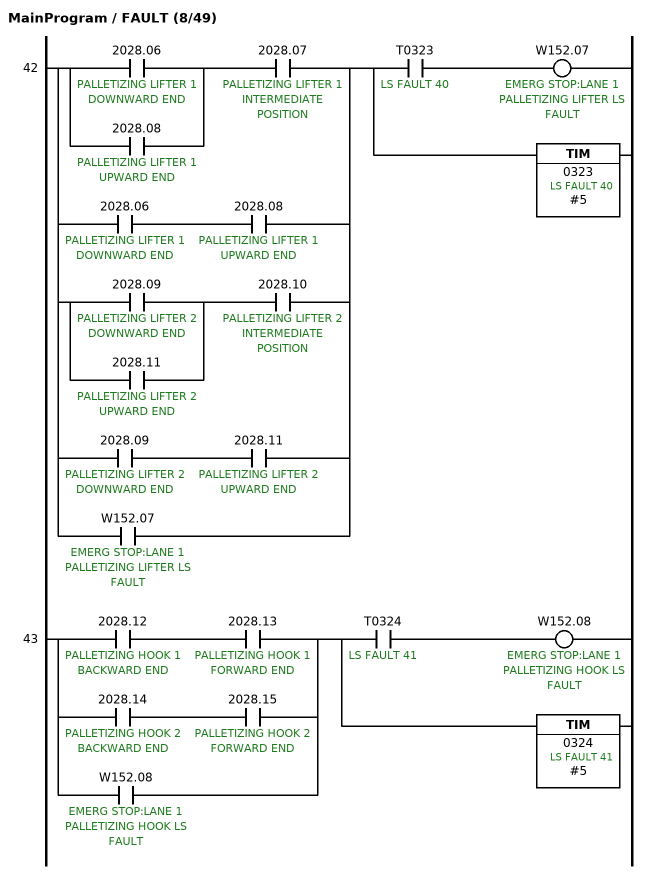
; rung 42
LD 2028.06  ; PALLETIZING LIFTER 1 DOWNWARD END
OR 2028.08  ; PALLETIZING LIFTER 1 UPWARD END
AND 2028.07  ; PALLETIZING LIFTER 1 INTERMEDIATE POSITION
LD 2028.06  ; PALLETIZING LIFTER 1 DOWNWARD END
AND 2028.08  ; PALLETIZING LIFTER 1 UPWARD END
ORLD
LD 2028.09  ; PALLETIZING LIFTER 2 DOWNWARD END
OR 2028.11  ; PALLETIZING LIFTER 2 UPWARD END
AND 2028.10  ; PALLETIZING LIFTER 2 INTERMEDIATE POSITION
ORLD
LD 2028.09  ; PALLETIZING LIFTER 2 DOWNWARD END
AND 2028.11  ; PALLETIZING LIFTER 2 UPWARD END
ORLD
OR W152.07  ; EMERG STOP:LANE 1 PALLETIZING LIFTER LS FAULT
OUT TR0
AND T0323  ; LS FAULT 40
OUT W152.07  ; EMERG STOP:LANE 1 PALLETIZING LIFTER LS FAULT
LD TR0
TIM 0323 #5  ; LS FAULT 40
; rung 43
LD 2028.12  ; PALLETIZING HOOK 1 BACKWARD END
AND 2028.13  ; PALLETIZING HOOK 1 FORWARD END
LD 2028.14  ; PALLETIZING HOOK 2 BACKWARD END
AND 2028.15  ; PALLETIZING HOOK 2 FORWARD END
ORLD
OR W152.08  ; EMERG STOP:LANE 1 PALLETIZING HOOK LS FAULT
OUT TR0
AND T0324  ; LS FAULT 41
OUT W152.08  ; EMERG STOP:LANE 1 PALLETIZING HOOK LS FAULT
LD TR0
TIM 0324 #5  ; LS FAULT 41

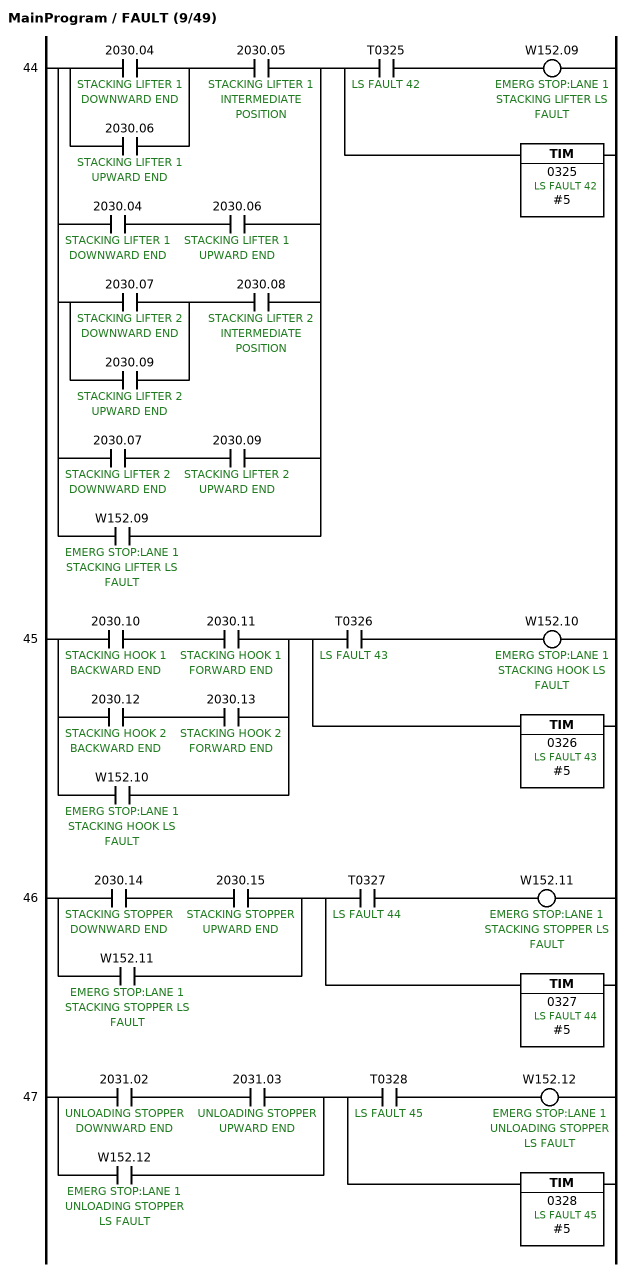
; rung 44
LD 2030.04  ; STACKING LIFTER 1 DOWNWARD END
OR 2030.06  ; STACKING LIFTER 1 UPWARD END
AND 2030.05  ; STACKING LIFTER 1 INTERMEDIATE POSITION
LD 2030.04  ; STACKING LIFTER 1 DOWNWARD END
AND 2030.06  ; STACKING LIFTER 1 UPWARD END
ORLD
LD 2030.07  ; STACKING LIFTER 2 DOWNWARD END
OR 2030.09  ; STACKING LIFTER 2 UPWARD END
AND 2030.08  ; STACKING LIFTER 2 INTERMEDIATE POSITION
ORLD
LD 2030.07  ; STACKING LIFTER 2 DOWNWARD END
AND 2030.09  ; STACKING LIFTER 2 UPWARD END
ORLD
OR W152.09  ; EMERG STOP:LANE 1 STACKING LIFTER LS FAULT
OUT TR0
AND T0325  ; LS FAULT 42
OUT W152.09  ; EMERG STOP:LANE 1 STACKING LIFTER LS FAULT
LD TR0
TIM 0325 #5  ; LS FAULT 42
; rung 45
LD 2030.10  ; STACKING HOOK 1 BACKWARD END
AND 2030.11  ; STACKING HOOK 1 FORWARD END
LD 2030.12  ; STACKING HOOK 2 BACKWARD END
AND 2030.13  ; STACKING HOOK 2 FORWARD END
ORLD
OR W152.10  ; EMERG STOP:LANE 1 STACKING HOOK LS FAULT
OUT TR0
AND T0326  ; LS FAULT 43
OUT W152.10  ; EMERG STOP:LANE 1 STACKING HOOK LS FAULT
LD TR0
TIM 0326 #5  ; LS FAULT 43
; rung 46
LD 2030.14  ; STACKING STOPPER DOWNWARD END
AND 2030.15  ; STACKING STOPPER UPWARD END
OR W152.11  ; EMERG STOP:LANE 1 STACKING STOPPER LS FAULT
OUT TR0
AND T0327  ; LS FAULT 44
OUT W152.11  ; EMERG STOP:LANE 1 STACKING STOPPER LS FAULT
LD TR0
TIM 0327 #5  ; LS FAULT 44
; rung 47
LD 2031.02  ; UNLOADING STOPPER DOWNWARD END
AND 2031.03  ; UNLOADING STOPPER UPWARD END
OR W152.12  ; EMERG STOP:LANE 1 UNLOADING STOPPER LS FAULT
OUT TR0
AND T0328  ; LS FAULT 45
OUT W152.12  ; EMERG STOP:LANE 1 UNLOADING STOPPER LS FAULT
LD TR0
TIM 0328 #5  ; LS FAULT 45

